FUNCTION FC_ProcessValue : DINT
VAR_INPUT
    nValue : DINT;
    bEnabled : BOOL;
END_VAR
VAR
    nResult : DINT;
END_VAR

nResult := 0;

IF bEnabled THEN
    IF nValue > 100 THEN
        nResult := 100;
    ELSIF nValue < 0 THEN
        nResult := 0;
    ELSE
        nResult := nValue;
    END_IF;
END_IF;

FC_ProcessValue := nResult;

END_FUNCTION

(* stored: Version 1.1.0.1
   POU FC_ProcessValue: Id {33333333-3333-3333-3333-333333333333}, SpecialFunc None *)
